// TIA Portal project "PLC-Lab-Rolltor-1500_PLCSim_V16_V18" (V18)

(* hardware
DEVICE "S71500/ET200MP-Station_1"  S7-1500 station
   slot 0: "Profilschiene_0"  Rack  6ES7 590-1***0-0AA0
   slot 0: "PS 60W 24/48/60VDC_1"  PS 60W 24/48/60VDC  6ES7 505-0RA00-0AB0  V1.0
   slot 1: "PLC_PlcLabProjektVorlage"  CPU 1511-1 PN  6ES7 511-1AK00-0AB0  V1.8
   slot 2: "DI 16x24VDC BA_1"  DI 16x24VDC BA  6ES7 521-1BH10-0AA0  V1.0
   slot 3: "AI 8xU/I/RTD/TC ST_1"  AI 8xU/I/RTD/TC ST  6ES7 531-7KF00-0AB0  V2.0
   slot 4: "AI 8xU/I/RTD/TC ST_2"  AI 8xU/I/RTD/TC ST  6ES7 531-7KF00-0AB0  V2.0
   slot 5: "AI 8xU/I/RTD/TC ST_3"  AI 8xU/I/RTD/TC ST  6ES7 531-7KF00-0AB0  V2.0
   slot 6: "AI 8xU/I/RTD/TC ST_4"  AI 8xU/I/RTD/TC ST  6ES7 531-7KF00-0AB0  V2.0
   slot 7: "AI 8xU/I/RTD/TC ST_5"  AI 8xU/I/RTD/TC ST  6ES7 531-7KF00-0AB0  V2.0
   slot 8: "AI 8xU/I/RTD/TC ST_6"  AI 8xU/I/RTD/TC ST  6ES7 531-7KF00-0AB0  V2.0
   slot 9: "AI 8xU/I/RTD/TC ST_7"  AI 8xU/I/RTD/TC ST  6ES7 531-7KF00-0AB0  V2.0
   slot 10: "AI 8xU/I/RTD/TC ST_8"  AI 8xU/I/RTD/TC ST  6ES7 531-7KF00-0AB0  V2.0
   slot 11: "AI 8xU/I/RTD/TC ST_9"  AI 8xU/I/RTD/TC ST  6ES7 531-7KF00-0AB0  V2.0
   slot 12: "AI 8xU/I/RTD/TC ST_10"  AI 8xU/I/RTD/TC ST  6ES7 531-7KF00-0AB0  V2.0
   slot 13: "AI 8xU/I/RTD/TC ST_11"  AI 8xU/I/RTD/TC ST  6ES7 531-7KF00-0AB0  V2.0
   slot 14: "AI 8xU/I/RTD/TC ST_12"  AI 8xU/I/RTD/TC ST  6ES7 531-7KF00-0AB0  V2.0
   slot 15: "AI 8xU/I/RTD/TC ST_13"  AI 8xU/I/RTD/TC ST  6ES7 531-7KF00-0AB0  V2.0
   slot 16: "AI 8xU/I/RTD/TC ST_14"  AI 8xU/I/RTD/TC ST  6ES7 531-7KF00-0AB0  V2.0
   slot 17: "AI 8xU/I/RTD/TC ST_15"  AI 8xU/I/RTD/TC ST  6ES7 531-7KF00-0AB0  V2.0
   slot 18: "AI 8xU/I/RTD/TC ST_16"  AI 8xU/I/RTD/TC ST  6ES7 531-7KF00-0AB0  V2.0
   slot 19: "AI 8xU/I/RTD/TC ST_17"  AI 8xU/I/RTD/TC ST  6ES7 531-7KF00-0AB0  V2.0
   slot 20: "AI 8xU/I/RTD/TC ST_18"  AI 8xU/I/RTD/TC ST  6ES7 531-7KF00-0AB0  V2.0
   slot 21: "AI 8xU/I/RTD/TC ST_19"  AI 8xU/I/RTD/TC ST  6ES7 531-7KF00-0AB0  V2.0
   slot 22: "AI 8xU/I/RTD/TC ST_20"  AI 8xU/I/RTD/TC ST  6ES7 531-7KF00-0AB0  V2.0
   slot 23: "AI 8xU/I/RTD/TC ST_21"  AI 8xU/I/RTD/TC ST  6ES7 531-7KF00-0AB0  V2.0
   slot 24: "AI 8xU/I/RTD/TC ST_22"  AI 8xU/I/RTD/TC ST  6ES7 531-7KF00-0AB0  V2.0
   slot 25: "AI 8xU/I/RTD/TC ST_23"  AI 8xU/I/RTD/TC ST  6ES7 531-7KF00-0AB0  V2.0
   slot 26: "AI 8xU/I/RTD/TC ST_24"  AI 8xU/I/RTD/TC ST  6ES7 531-7KF00-0AB0  V2.0
   slot 27: "AI 8xU/I/RTD/TC ST_25"  AI 8xU/I/RTD/TC ST  6ES7 531-7KF00-0AB0  V2.0
   slot 28: "AI 8xU/I/RTD/TC ST_26"  AI 8xU/I/RTD/TC ST  6ES7 531-7KF00-0AB0  V2.0
   slot 29: "AI 8xU/I/RTD/TC ST_27"  AI 8xU/I/RTD/TC ST  6ES7 531-7KF00-0AB0  V2.0
   slot 30: "AI 8xU/I/RTD/TC ST_28"  AI 8xU/I/RTD/TC ST  6ES7 531-7KF00-0AB0  V2.0
   slot 31: "AI 8xU/I/RTD/TC ST_29"  AI 8xU/I/RTD/TC ST  6ES7 531-7KF00-0AB0  V2.0
*)

// ===== PLC "PLC_PlcLabProjektVorlage"  CPU 1511-1 PN =====

VAR_GLOBAL   // PLC tag table "Standard-Variablentabelle"
   "S1" AT %E20.0 : Bool;   // Taster "Tor zufahren" (no)
   "S2" AT %E20.1 : Bool;   // Taster "Tor auffahren" (no)
   "Clock_1.25Hz" AT %M0.4 : Bool;   // Taktmerker mit 1,25 Hz
   "S3" AT %E20.2 : Bool;   // Schlüsselschalter (no)
   "S5" AT %E20.3 : Bool;   // Taster "Stopp" (nc)
   "S0" AT %E20.4 : Bool;   // Schalter "Not-Halt" (nc)
   "S8 (B8)" AT %E20.5 : Bool;   // Endlage "Tor ist zu" (nc)
   "S9 (B9)" AT %E20.6 : Bool;   // Endlage "Tor ist auf" (nc)
   "B1" AT %E20.7 : Bool;   // Lichtschranke (no)
   "K1 (Q1)" AT %A20.0 : Bool;   // Schütz "Tor zufahren"
   "K2 (Q2)" AT %A20.1 : Bool;   // Schütz "Tor auffahren"
   "V1 (P1)" AT %A20.2 : Bool;   // Melder "Tor fährt"
   "H8 (P8)" AT %A20.3 : Bool;   // Tonmelder "Tor fährt"
   "P3" AT %A20.4 : Bool;   // Leuchttaster "Tor zufahren"
   "P4" AT %A20.5 : Bool;   // Leuchttaster "Tor auffahren"
   "P5" AT %A20.6 : Bool;   // Leuchttaster "Stopp"
END_VAR

DATA_BLOCK "rolltor_DB"   // DB1
{ S7_Optimized_Access := 'TRUE' }
VERSION : 0.1
// stored: InstanceOfName rolltor
"rolltor"
BEGIN
END_DATA_BLOCK

// folder: System blocks/Program resources

DATA_BLOCK "IEC_Timer_0_DB"   // DB2
{ S7_Optimized_Access := 'TRUE' }
AUTHOR : Simatic
FAMILY : IEC
NAME : IEC_TMR
VERSION : 1.0
// stored: InstanceOfName IEC_TIMER
"IEC_TIMER"
BEGIN
END_DATA_BLOCK

DATA_BLOCK "IEC_Timer_0_DB_1"   // DB3
{ S7_Optimized_Access := 'TRUE' }
AUTHOR : Simatic
FAMILY : IEC
NAME : IEC_TMR
VERSION : 1.0
// stored: InstanceOfName IEC_TIMER
"IEC_TIMER"
BEGIN
END_DATA_BLOCK

// folder: (top level)

FUNCTION_BLOCK "rolltor"   // FB1, FBD
{ S7_Optimized_Access := 'TRUE' }
VERSION : 0.1
   VAR_INPUT
      tasterAuf : Bool;
      tasterZu : Bool;
      schluessel : Bool;
      tasterStop : Bool;
      "not-halt" : Bool;
      clock : Bool;
      sensorAufEndlage : Bool;
      sensorZuEndlage : Bool;
      lichtschranke : Bool;
   END_VAR
   VAR_OUTPUT
      motorAuf : Bool;
      motorZu : Bool;
      leuchteStop : Bool;
      leuchteTasterAuf : Bool;
      leuchteTasterZu : Bool;
      tonFahr : Bool;
      melderFahr : Bool;
   END_VAR
   VAR
      merkeAuf : Bool;
      merkeZu : Bool;
   END_VAR
BEGIN

REGION Network 1
   // Rolltor Auf
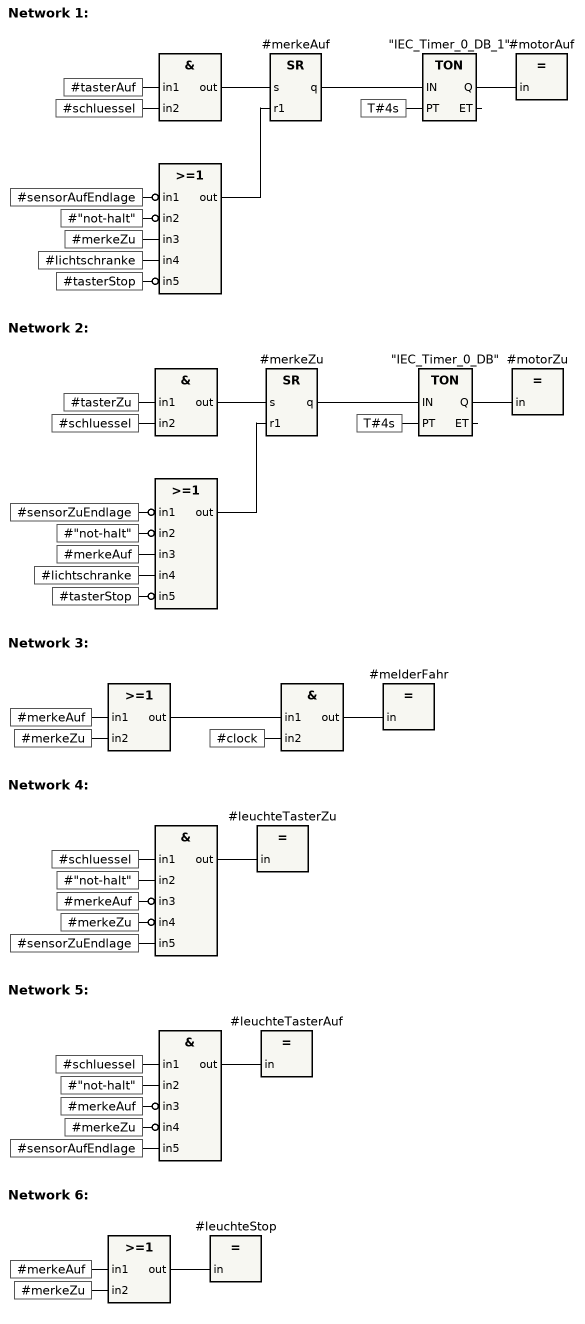
   IF #tasterAuf AND #schluessel THEN
       #merkeAuf := TRUE;   // SR flip-flop
   END_IF;
   IF NOT #sensorAufEndlage OR NOT #"not-halt" OR #merkeZu OR #lichtschranke OR NOT #tasterStop THEN
       #merkeAuf := FALSE;
   END_IF;
   "IEC_Timer_0_DB_1".TON(IN := #merkeAuf, PT := T#4s);
   #motorAuf := "IEC_Timer_0_DB_1".Q;
END_REGION

REGION Network 2
   // Rolltor Zu
   IF #tasterZu AND #schluessel THEN
       #merkeZu := TRUE;   // SR flip-flop
   END_IF;
   IF NOT #sensorZuEndlage OR NOT #"not-halt" OR #merkeAuf OR #lichtschranke OR NOT #tasterStop THEN
       #merkeZu := FALSE;
   END_IF;
   "IEC_Timer_0_DB".TON(IN := #merkeZu, PT := T#4s);
   #motorZu := "IEC_Timer_0_DB".Q;
END_REGION

REGION Network 3
   // Leuchten
   #melderFahr := (#merkeAuf OR #merkeZu) AND #clock;
END_REGION

REGION Network 4
   // Leuchte zu
   #leuchteTasterZu := #schluessel AND #"not-halt" AND NOT #merkeAuf AND NOT #merkeZu AND #sensorZuEndlage;
END_REGION

REGION Network 5
   // Leuchte Auf
   #leuchteTasterAuf := #schluessel AND #"not-halt" AND NOT #merkeAuf AND NOT #merkeZu AND #sensorAufEndlage;
END_REGION

REGION Network 6
   // Leuchte Stop
   #leuchteStop := #merkeAuf OR #merkeZu;
END_REGION
END_FUNCTION_BLOCK

FUNCTION "MHJ-PLC-Lab-Function-S71500" : Void   // FC1, SCL
{ S7_Optimized_Access := 'TRUE' }
VERSION : 0.1
   VAR_INPUT
      MinDiByte : Int;
      MaxDiByte : Int;
   END_VAR
   VAR_TEMP
      Value : Byte;
      ForCounter : Int;
      MaxDiByteTemp : Int;
      MinDiByteTemp : Int;
   END_VAR
   VAR CONSTANT
      Value_01_DW : DWord := 16#1223_5486;
      Value_02_DW : DWord := 16#A6C9_D1F5;
   END_VAR
BEGIN

   #Value:=PEEK(area := 16#82,
        dbNumber := 0,
        byteOffset := 511);
   #Value := #Value + 1;

   POKE(area := 16#82,
        dbNumber := 0,
        byteOffset := 511,
        value := #Value);

   POKE(area := 16#82,
        dbNumber := 0,
        byteOffset := 1016,
        value := #Value_01_DW);
   POKE(area := 16#82,
        dbNumber := 0,
        byteOffset := 1020,
        value := #Value_02_DW);

   #MaxDiByteTemp := 462;
   IF #MaxDiByte < 463 THEN
       #MaxDiByteTemp := #MaxDiByte;
   END_IF;

   #MinDiByteTemp := 0;
   IF #MaxDiByteTemp >= #MinDiByte & #MinDiByte >= 0 THEN
       #MinDiByteTemp := #MinDiByte;
   END_IF;

   FOR #ForCounter := #MinDiByteTemp TO #MaxDiByteTemp DO
       #Value := PEEK(area := 16#1,
                      dbNumber := 0,
                      byteOffset := #ForCounter);
       POKE(area := 16#81,
            dbNumber := 0,
            byteOffset := #ForCounter,
            value := #Value);
   END_FOR;

   #Value := PEEK(area := 16#1,
                  dbNumber := 0,
                  byteOffset := 512);
   POKE(area := 16#82,
        dbNumber := 0,
        byteOffset := 512,
        value := #Value);
END_FUNCTION

ORGANIZATION_BLOCK "Main"   // OB1, FBD, ProgramCycle
TITLE = "Main Program Sweep (Cycle)"
{ S7_Optimized_Access := 'TRUE' }
VERSION : 0.1
   VAR_INPUT
      Initial_Call : Bool;   // Initial call of this OB
      Remanence : Bool;   // =True, if remanent data are available
   END_VAR
BEGIN

REGION Network 1
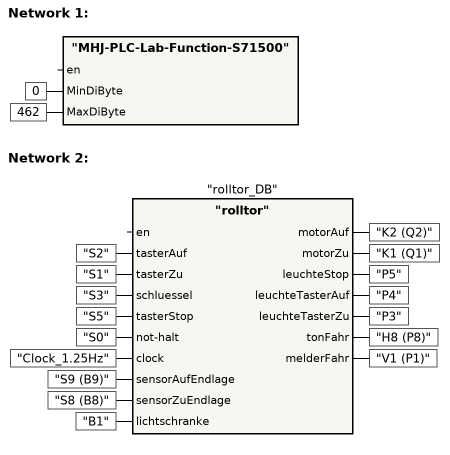
   "MHJ-PLC-Lab-Function-S71500"(MinDiByte := 0, MaxDiByte := 462);
END_REGION

REGION Network 2
   "rolltor_DB"(tasterAuf := "S2",   // "rolltor"
                tasterZu := "S1",
                schluessel := "S3",
                tasterStop := "S5",
                "not-halt" := "S0",
                clock := "Clock_1.25Hz",
                sensorAufEndlage := "S9 (B9)",
                sensorZuEndlage := "S8 (B8)",
                lichtschranke := "B1",
                motorAuf => "K2 (Q2)",
                motorZu => "K1 (Q1)",
                leuchteStop => "P5",
                leuchteTasterAuf => "P4",
                leuchteTasterZu => "P3",
                tonFahr => "H8 (P8)",
                melderFahr => "V1 (P1)");
END_REGION
END_ORGANIZATION_BLOCK